FUNCTION_BLOCK FB_LinkDataDWord EXTENDS FB_LinkDevice
VAR		
	ControlData		AT %Q* : DWORD; //{simulation-interface}
	StatusData		AT %I* : DWORD; //{simulation-interface}	
END_VAR

SUPER^();

METHOD INTERNAL GetLinkControlData : DWORD
GetLinkControlData := ControlData;
END_METHOD

METHOD INTERNAL SetLinkStatusData : BOOL
VAR_INPUT
	nStatusData : DWORD;
END_VAR
StatusData := nStatusData;
END_METHOD

END_FUNCTION_BLOCK

(* stored: Version 1.1.0.1, ProductVersion 3.1.4024.12
   POU FB_LinkDataDWord: Id {6640c605-874d-0b5b-3d68-62428ba9b094}, SpecialFunc None
   Method GetLinkControlData: Id {741520f1-4770-0983-0fe1-555395da09ab}
   Method SetLinkStatusData: Id {c74d0794-b847-0043-3a61-8919b309200a} *)
